TYPE Mat43 : ARRAY[1..4, 1..3] OF LREAL; END_TYPE

(* stored: Version 1.1.0.1, ProductVersion 3.1.4024.12
   DUT Mat43: Id {79a3f313-e557-45cb-ab20-e3820638f803} *)
